(* IEC 61131-3 sources: ICSQuartz/benchmarks/oscat_basic_replace_all/src, 1 file *)

(* ---- program.st ---- *)
PROGRAM PLC_PRG
VAR_INPUT
    in_STR: STRING;
    in_SRC: STRING;
    in_REP: STRING;
END_VAR

REPLACE_ALL(in_STR, in_SRC, in_REP);

END_PROGRAM
